(* CODESYS project Tags.library
   Company: _
   DefaultNamespace: Tags
   Title: Tags
   Placeholder: _Tags
   Author: Krystian Lis et al.
   Description: Universal identification.
   Version: 1.0.0

Project tree, tasks and I/O mapping:
  libraries: Debug, * (_); Results, * (_); Strings, * (_); Tc2_Standard, * (Beckhoff Automation GmbH)
  Tag/
    function block A_Tag [ST]: FB_Init, ToDebug
    interface I_Tag: Cache, GetId, Join, Leave, Option, Owner, Self
    interface I_TagCmp: AndIf, Default, IsErr, IsOk, Match, MatchId, MatchPrtId, OrIf, Set, XorIf
    interface I_Tagged: Tag
    interface I_TagOwner
    function block Tag [ST]: Cache, FB_init, GetId, Join, Leave, Option, Owner, Self, ToDebug
    function block TagCmp [ST]: _self, AndIf, Default, IsErr, IsOk, Match, MatchId, MatchPrtId, OrIf, Set, XorIf
    function block TagOwner [ST]: Self
*)

// Tag/A_Tag
FUNCTION_BLOCK A_Tag IMPLEMENTS Debug.I_Debug

//FB_Init is always available implicitly and it is used primarily for initialization.
//The return value is not evaluated. For a specific influence, you can also declare the
//methods explicitly and provide additional code there with the standard initialization
//code. You can evaluate the return value.
METHOD FB_Init: BOOL
VAR_INPUT
    bInitRetains: BOOL; // TRUE: the retain variables are initialized (reset warm / reset cold)
    bInCopyCode: BOOL;  // TRUE: the instance will be copied to the copy code afterward (online change)
	
	iTag			: I_Tag;
	refTag			: REFERENCE TO I_Tag;
END_VAR
IF NOT __ISVALIDREF(refTag) THEN
	Debug.DebugMsg(THIS^, ': Ref = 0!');
	RETURN;
END_IF

IF iTag = 0 THEN
	Debug.DebugMsg(THIS^, ': Itf = 0!');
	RETURN;
END_IF

IF refTag <> 0 THEN
	Debug.DebugMsg(THIS^, ': Ref itf should be unassigned!');
	RETURN;
END_IF

refTag := iTag;
END_METHOD

METHOD ToDebug : Debug.I_Debug
ToDebug := THIS^;
END_METHOD

END_FUNCTION_BLOCK

// Tag/I_Tag
INTERFACE I_Tag EXTENDS Debug.I_Debug

PROPERTY Cache : UDINT
GET
END_GET
END_PROPERTY

METHOD GetId : Strings.Str
VAR_INPUT
END_VAR
END_METHOD

METHOD Join : Results.Result
VAR_INPUT
	iOwner		: I_TagOwner;
	nCache		: UDINT;
END_VAR
END_METHOD

METHOD Leave : Results.Result
VAR_INPUT
	iOwner		: I_TagOwner;
END_VAR
END_METHOD

PROPERTY Option : Strings.Str
GET
END_GET
END_PROPERTY

PROPERTY Owner : I_TagOwner
GET
END_GET
END_PROPERTY

PROPERTY Self : I_Tag
GET
END_GET
END_PROPERTY

END_INTERFACE

// Tag/I_TagOwner
INTERFACE INTERNAL I_TagOwner

END_INTERFACE

// Tag/I_TagCmp
INTERFACE INTERNAL I_TagCmp

METHOD AndIf : I_TagCmp
VAR_INPUT
	bCondition: BOOL;
END_VAR
END_METHOD

METHOD Default : BOOL
END_METHOD

METHOD IsErr : BOOL
END_METHOD

METHOD IsOk : BOOL
END_METHOD

METHOD Match : I_TagCmp
VAR_INPUT
	iOther: I_Tag;
END_VAR
END_METHOD

METHOD MatchId : I_TagCmp
VAR_INPUT
	sOtherId	: Strings.Str;
END_VAR
END_METHOD

METHOD MatchPrtId : I_TagCmp
VAR_INPUT
	sPartialId		: Strings.Str;
END_VAR
END_METHOD

METHOD OrIf : I_TagCmp
VAR_INPUT
	bCondition: BOOL;
END_VAR
END_METHOD

METHOD Set : I_TagCmp
VAR_INPUT
	iBaseTag	: I_Tag;
END_VAR
END_METHOD

METHOD XorIf : I_TagCmp
VAR_INPUT
	bCondition: BOOL;
END_VAR
END_METHOD

END_INTERFACE

// Tag/I_Tagged
INTERFACE I_Tagged

PROPERTY Tag : I_Tag
GET
END_GET
END_PROPERTY

END_INTERFACE

// Tag/Tag
{attribute 'reflection'}
FUNCTION_BLOCK Tag IMPLEMENTS I_Tag
VAR
	{attribute 'instance-path'} 
    {attribute 'noinit'} 
	_sId			: Strings.Str;
	_nOptionPos		: USINT;
	_nOptionLen		: USINT;
	_nCache			: UDINT;
	_iOwner			: I_TagOwner;
END_VAR

PROPERTY Cache : UDINT
GET
Cache := _nCache;
END_GET
END_PROPERTY

METHOD FB_init : BOOL
VAR_INPUT
	bInitRetains : BOOL; // if TRUE, the retain variables are initialized (warm start / cold start)
	bInCopyCode : BOOL;  // if TRUE, the instance afterwards gets moved into the copy code (online change)
END_VAR
VAR
	i				: INT;
END_VAR
// Delete this name
FOR i := Tc2_Standard.LEN(_sId) TO 1 BY -1 DO
	IF Tc2_Standard.MID(_sId, 1, i) = '.' THEN
		_sId := Tc2_Standard.LEFT(_sId, i - 1);
		EXIT;
	END_IF
END_FOR

// Delete project name
FOR i := 1 TO Tc2_Standard.LEN(_sId) DO
	IF Tc2_Standard.MID(_sId, 1, i) = '.' THEN
		_sId := Tc2_Standard.DELETE(_sId, i, 1);
		EXIT;
	END_IF
END_FOR

// Delete plc name
FOR i := 1 TO Tc2_Standard.LEN(_sId) DO
	IF Tc2_Standard.MID(_sId, 1, i) = '.' THEN
		_sId := Tc2_Standard.DELETE(_sId, i, 1);
		EXIT;
	END_IF
END_FOR
END_METHOD

METHOD GetId : Strings.Str
VAR_INPUT
END_VAR
IF _nOptionPos <> 0 THEN
	GetId := Tc2_Standard.DELETE(_sId, _nOptionLen, _nOptionPos); 
ELSE
	GetId := _sId;
END_IF
END_METHOD

METHOD Join : Results.Result
VAR_INPUT
	iOwner		: I_TagOwner;
	nCache		: UDINT;
END_VAR
IF iOwner = 0 THEN
	Join := Results.Err.Itf0;
	RETURN;
END_IF

IF _iOwner <> 0 THEN
	Join := Results.Err.ItfEq;
	RETURN;
END_IF

_iOwner := iOwner;
_nCache := nCache;
Join := Results.Ok;
END_METHOD

METHOD Leave : Results.Result
VAR_INPUT
	iOwner		: I_TagOwner;
END_VAR
IF iOwner = 0 THEN
	Leave := Results.Err.Itf0;
	RETURN;
END_IF

IF _iOwner <> iOwner THEN
	Leave := Results.Err.ItfEq;
	RETURN;
END_IF

_iOwner := 0;
Leave := Results.Ok;
END_METHOD

PROPERTY Option : Strings.Str
GET
VAR
	i				: INT;
END_VAR
IF _nOptionPos <> 0 THEN
	Option := Tc2_Standard.DELETE(_sId, _nOptionPos, 1); 
ELSE
	Option := '';
END_IF
END_GET
SET
VAR
	nCase		: USINT;
END_VAR
IF Option <> '' THEN
    _nOptionLen := INT_TO_USINT(Tc2_Standard.LEN(Option));    
    IF _nOptionPos <> 0 THEN
        _sId := Tc2_Standard.LEFT(_sId, _nOptionPos);
        _sId := Tc2_Standard.CONCAT(_sId, Option);
    ELSE
        // The option does not exist, so we append it
        _nOptionPos := INT_TO_USINT(Tc2_Standard.LEN(_sId) + 1);
        _sId := Tc2_Standard.CONCAT(_sId, '.');
        _sId := Tc2_Standard.CONCAT(_sId, Option);
    END_IF
ELSIF _nOptionPos <> 0 THEN
    _sId := Tc2_Standard.LEFT(_sId, _nOptionPos - 1);
    _nOptionPos := 0;
END_IF
END_SET
END_PROPERTY

PROPERTY Owner : I_TagOwner
GET
Owner := _iOwner;
END_GET
END_PROPERTY

PROPERTY Self : I_Tag
GET
Self := THIS^;
END_GET
END_PROPERTY

METHOD ToDebug : Debug.I_Debug
ToDebug := THIS^;
END_METHOD

END_FUNCTION_BLOCK

// Tag/TagCmp
FUNCTION_BLOCK TagCmp IMPLEMENTS I_TagCmp
VAR
	_iBaseTag		: I_Tag;
	_eResult		: Results.Result;
	_bLock			: BOOL;
END_VAR

PROPERTY PRIVATE _self : I_TagCmp
GET
VAR
	_this : I_TagCmp := THIS^;
END_VAR
_self := _this;
END_GET
END_PROPERTY

METHOD AndIf : I_TagCmp
VAR_INPUT
	bCondition: BOOL;
END_VAR
AndIf := _self;

IF _bLock THEN
	RETURN;
END_IF

IF _eResult = Results.Ok AND_THEN bCondition THEN
	_eResult := Results.Ok;
END_IF
END_METHOD

METHOD Default : BOOL
IF _bLock THEN
	RETURN;
END_IF

IF _eResult <> Results.None THEN
	RETURN;
END_IF

_bLock := TRUE;
Default := TRUE;
END_METHOD

METHOD IsErr : BOOL
IF _bLock THEN
	RETURN;
END_IF

IF _eResult >= 0 THEN
	RETURN;
END_IF

_bLock := TRUE;
IsErr := TRUE;
END_METHOD

METHOD IsOk : BOOL
IF _bLock THEN
	RETURN;
END_IF

IF _eResult <> Results.Ok THEN
	RETURN;
END_IF

_bLock := TRUE;
IsOk := TRUE;
END_METHOD

METHOD Match : I_TagCmp
VAR_INPUT
	iOther: I_Tag;
END_VAR
Match := _self;

IF _bLock THEN
	RETURN;
END_IF

CASE _eResult OF
	Results.Ok,
	Results.None:
		IF iOther = _iBaseTag THEN
			_eResult := Results.Ok;
		END_IF
END_CASE
END_METHOD

METHOD MatchId : I_TagCmp
VAR_INPUT
	sOtherId	: Strings.Str;
END_VAR
MatchId := _self;

IF _bLock THEN
	RETURN;
END_IF

CASE _eResult OF
	Results.Ok,
	Results.None:
		IF sOtherId <> '' AND_THEN _iBaseTag.GetId() = sOtherId THEN
			_eResult := Results.Ok;
		END_IF
END_CASE
END_METHOD

METHOD MatchPrtId : I_TagCmp
VAR_INPUT
	sPartialId		: Strings.Str;
END_VAR
MatchPrtId := _self;

IF _bLock THEN
	RETURN;
END_IF

CASE _eResult OF
	Results.Ok,
	Results.None:
		IF sPartialId <> '' AND_THEN (Tc2_Standard.RIGHT(_iBaseTag.GetId(), Tc2_Standard.LEN(sPartialId)) = sPartialId) THEN
			_eResult := Results.Ok;
		END_IF
END_CASE
END_METHOD

METHOD OrIf : I_TagCmp
VAR_INPUT
	bCondition: BOOL;
END_VAR
OrIf := _self;

IF _bLock THEN
	RETURN;
END_IF

IF _eResult = Results.Ok OR_ELSE bCondition THEN
	_eResult := Results.Ok;
END_IF
END_METHOD

METHOD Set : I_TagCmp
VAR_INPUT
	iBaseTag	: I_Tag;
END_VAR
_iBaseTag := iBaseTag;
_eResult := Results.None;
_bLock := FALSE;

IF iBaseTag = 0 THEN
	_eResult := Results.Err.Itf0;
END_IF

Set := _self;
END_METHOD

METHOD XorIf : I_TagCmp
VAR_INPUT
	bCondition: BOOL;
END_VAR
XorIf := _self;

IF _bLock THEN
	RETURN;
END_IF

IF _eResult = Results.Ok XOR bCondition THEN
	_eResult := Results.Ok;
END_IF
END_METHOD

END_FUNCTION_BLOCK

// Tag/TagOwner
FUNCTION_BLOCK TagOwner IMPLEMENTS I_TagOwner;

PROPERTY Self : I_TagOwner
GET
Self := THIS^;
END_GET
END_PROPERTY

END_FUNCTION_BLOCK
